TYPE ST_COUPLER_DETECT_SETTINGS :
STRUCT
//	startPoint:		TcVnPoint2_REAL := [1000, 550];
//	endPoint:		TcVnPoint2_REAL := [550, 1000];
	
//	minStrength:	REAL := 45;
//	searchLines:	UDINT := 5;
	
END_STRUCT
END_TYPE

(* stored: Version 1.1.0.1
   DUT ST_COUPLER_DETECT_SETTINGS: Id {66f465b5-842f-4184-b3b1-184b450f3a9f} *)
